FUNCTION_BLOCK FB_ZLevelSensor EXTENDS FB_MzTool
VAR_INPUT
END_VAR
VAR_OUTPUT
END_VAR
VAR
	rCurrentZMeasPos	: REAL;
	rZMeasPosOffset		: REAL;
END_VAR

SUPER^();	//FB_MzTool aufrufen

//Prozessdaten aktualisieren
IF pZAxisRef > 0 THEN
	stProcessData.n32Data[7] := BOOL_TO_DINT(pZAxisRef^.stInput.nToolState.1);
END_IF
aObjProcData[nNotifyId] := stProcessData;

ACTION A_Reset:
nStateA_ResetSpec := 80;
SUPER^.A_Reset();
END_ACTION

METHOD FB_init : BOOL
VAR_INPUT
	bInitRetains : BOOL; // if TRUE, the retain variables are initialized (warm start / cold start)
	bInCopyCode : BOOL;  // if TRUE, the instance afterwards gets moved into the copy code (online change)
END_VAR
eObjectType := E_ObjectType.OBJECTTYPE_ZSensor;
eObjectGroup := E_ObjectGroup.OBJECTGROUP_MzTool OR E_ObjectGroup.OBJECTGROUP_Device;
END_METHOD

METHOD M_AddChild : ERRORID
VAR_INPUT
	pObject : POINTER TO FB_Object;
	nSlotNr	: UINT;
	nIndex 	: INT;
END_VAR
//Kann keine Objekte aufnehmen
M_AddChild := E_ErrorIdObjMgmt.ERRORID_ObjectCanNotTakeChilds;
END_METHOD

METHOD M_CheckAction : ERRORID
VAR_INPUT
	refActionData 	: REFERENCE TO ST_ActionData;
	pCorrelObject	: POINTER TO FB_Object;
END_VAR

VAR
	eMeasureMode : E_MeasureMode;
	pInkStation	 : POINTER TO FB_InkStation;
END_VAR
CASE refActionData.eAction OF
	E_Action.ACTION_MeasureTool:
		//ZSensor montiert?
		IF NOT P_bSensorMounted THEN
			M_CheckAction := E_ErrorIdCmd.ERRORID_ZSensorNotMounted;
		END_IF
		//MeasureMode auswerten
		eMeasureMode := DINT_TO_USINT(refActionData.aParams[1]);
		IF eMeasureMode = E_MeasureMode.MEAS_MODE_Auto THEN	//Target muss passend sein
			CASE fbObjectDirectory.M_GetObjType(refActionData.nTarget) OF
				E_ObjectType.OBJECTTYPE_InkStation:
					pInkStation := fbObjectDirectory.M_GetObjPointer(refActionData.nTarget);
					//Inkstation offen?
					IF (pInkStation^.P_eCoverState <> E_OpClState.Open) THEN
						M_CheckAction := E_ErrorIdCmd.ERRORID_InkStationNotOpen;
						RETURN;
					END_IF
					//Inkstation im Stillstand?
					IF(pInkStation^.P_nCurrentSpinSpeed <> 0) THEN
						M_CheckAction := E_ErrorIdCmd.ERRORID_InkStationIsStillSpinning;
						RETURN;
					END_IF
				E_ObjectType.OBJECTTYPE_DryPad,
				E_ObjectType.OBJECTTYPE_Slide,
				//E_ObjectType.OBJECTTYPE_Wafer,
				E_ObjectType.OBJECTTYPE_Point:
				//Do nothing
			ELSE
				M_CheckAction := E_ErrorIdCmd.ERRORID_UnsuitableTarget;
				RETURN;
			END_CASE
		
		ELSIF eMeasureMode = E_MeasureMode.MEAS_MODE_SemiAuto THEN	//Target muss erst ermittelt werden
			//nMeasToolTargetIdx := aI_MzTool[nMeasToolMzToolIdx].M_GetCurrentTargetIdx();
			//passendes Target gefunden?
			(*IF NOT (aI_Target[nMeasToolTargetIdx].P_eObjectType = E_ObjectType.OBJECTTYPE_Slide OR 
				aI_Target[nMeasToolTargetIdx].P_eObjectType = E_ObjectType.OBJECTTYPE_DryPad OR
				aI_Target[nMeasToolTargetIdx].P_eObjectType = E_ObjectType.OBJECTTYPE_Wafer) THEN
				M_ExeAction := E_ErrorIdCmd.ERRORID_InvalidTarget;
				RETURN;					
			END_IF*)
			;
		ELSE
			M_CheckAction := E_ErrorIdCmd.ERRORID_InvalidMeasureMode;
			RETURN;
		END_IF	
ELSE
	M_CheckAction := SUPER^.M_CheckAction(refActionData, pCorrelObject);	
END_CASE
END_METHOD

METHOD M_SetAllProps : ERRORID
VAR_INPUT
	refCmdData : REFERENCE TO  ST_CmdData;
END_VAR

VAR
	pExtruder : POINTER TO FB_Extruder;
END_VAR
IF pParentMzTool^.P_eObjectType = E_ObjectType.OBJECTTYPE_SinglePiezoHolder THEN
	;	
ELSIF pParentMzTool^.P_eObjectType = E_ObjectType.OBJECTTYPE_Extruder THEN
	pExtruder := pParentMzTool;
	IF pExtruder^.P_eExtruderType <> E_ExtruderType.SyringeExtruder1 THEN
		M_SetAllProps := E_ErrorIdObjMgmt.ERRORID_InvalidParentMzTool;
		RETURN;	
	END_IF
ELSE
	M_SetAllProps := E_ErrorIdObjMgmt.ERRORID_InvalidParentMzTool;
	RETURN;	
END_IF

M_SetAllProps := SUPER^.M_SetAllProps(refCmdData);
END_METHOD

PROPERTY P_bCollFree : BOOL
GET
VAR
	st3DPoint 		: ST_3DPoint;
END_VAR
//wenn Z-Stift nicht montiert, dann kollisionsfrei
IF pZAxisRef^.stInput.nToolState.1 THEN
	P_bCollFree := SUPER^.P_bCollFree;
ELSE
	P_bCollFree := TRUE;
END_IF
END_GET
END_PROPERTY

PROPERTY P_bSensorMounted : BOOL
GET
IF pParentMzTool^.P_eObjectType = E_ObjectType.OBJECTTYPE_SinglePiezoHolder OR pParentMzTool^.P_eObjectType = E_ObjectType.OBJECTTYPE_Extruder THEN
	P_bSensorMounted := pZAxisRef^.stInput.nToolState.1;	
END_IF
END_GET
END_PROPERTY

PROPERTY P_rToolRadius : REAL
GET
VAR
	stDim : ST_3DDimension;
END_VAR
P_rToolRadius := 1500.0;
END_GET
END_PROPERTY

END_FUNCTION_BLOCK

(* stored: Version 1.1.0.1, ProductVersion 3.1.4024.15
   POU FB_ZLevelSensor: Id {fbda1e44-eb3b-40cc-ae60-715d8a0464c4}, SpecialFunc None
   Action A_Reset: Id {df4bcb09-4b44-484d-9ff4-37b3c4eecaf1}
   Method FB_init: Id {772740e4-1f67-4d17-b236-730d3374c0a5}
   Method M_AddChild: Id {747778e0-2575-4016-80b3-3c449bb1c9c2}
   Method M_CheckAction: Id {cf00a1fc-8a89-4e50-9e96-695196791137}
   Method M_SetAllProps: Id {f9bfc7a9-f3f4-48ef-a67c-31066ee7c4ec}
   Property P_bCollFree: Id {7cd3c43f-9bd4-458b-a46a-36d68ca2554d}
   Get Get: Id {fd2dba47-00f5-40f9-bca3-7ba16e674bf5}
   Property P_bSensorMounted: Id {21c421d0-2f76-4f85-8729-4a3e6a44f849}
   Get Get: Id {ba9ccc56-3b8b-4364-95ea-345fbe8425ae}
   Property P_rToolRadius: Id {5f79db89-bcb6-4b12-afe1-0c78e489bca1}
   Get Get: Id {359ef27e-6ced-4be0-913e-1cd936e03e28} *)
